// TIA Portal V18 export
TYPE "UDT_Gripper_Fixture_Codes"
// =================================================================================
//  OTHER UDTs (Grippers, Process, etc. - Unchanged from previous correct versions)
//  =================================================================================
   STRUCT
      "JAW TOOLING LEFT" : String[128];
      "JAW TOOLING RIGHT" : String[128];
      "SHAFT CLAMPING LEFT" : String[128];
      "SHAFT CLAMPING RIGHT" : String[128];
   END_STRUCT;
END_TYPE
